(* PLC project v0.6.02_RefactorGateAndTest.project, CODESYS CODESYS V3.5 SP19 Patch 1 *)
(* stored: creationDateTime 2026-08-11T18:19:14.763505, modificationDateTime 2026-08-11T18:19:14.763505 *)

(* ═══════════════════════════════════════════════════════════════ 🔌 ST_ContactorCheck — Double vérification commande/retour contacteur ─────────────────────────────────────────────────────────────── 📄 Doc métier : DOC/AF/AF_Partie-02_Architecture_Programme_v3.1.md §3, DOC/AF/AF_Partie-03_Contrats_Composants_v2.1.md §2 Utilisé par FB_Brake (frein) et FB_Winch (contacteurs de sens) pour détecter un collage / une absence de fermeture d'un contacteur de puissance, au-delà d'un délai de cohérence (FeedbackTimeout du FB appelant). ═══════════════════════════════════════════════════════════════ *)
TYPE ST_ContactorCheck : STRUCT
  Command : BOOL;  (* Ordre envoyé au contacteur (TRUE = fermé/actif) *)
  Feedback : BOOL;  (* Retour d'état câblé (TRUE = effectivement fermé) *)
  StuckClosed : BOOL;  (* Diag : commande OFF mais retour ON depuis trop longtemps → PowerCutOff *)
  StuckOpen : BOOL;  (* Diag : commande ON mais retour OFF depuis trop longtemps *)
END_STRUCT;
END_TYPE
